// TIA Portal V19 export
TYPE "LAF_typeXXXEmXParametersInterface"
// stored: Access Published
   STRUCT
      configuration : "LAF_typeXXXParameters";
      commands : "LBC_typeInterfaceCommands";
      monitoring { S7_SetPoint := 'True'} : "LAF_typeXXXProcessValues";
   END_STRUCT;
END_TYPE
